(* IEC 61131-3 sources: test/Class/Sfc_Client_Splitter_4, 1 file *)

(* ---- Sfc_Client_Splitter_4.st ---- *)
(*!
<Class
	Name               = "Sfc_Client_Splitter_4"
	Revision           = "1.2"
	RealtimeTask       = "false"
	CyclicTask         = "false"
	BackgroundTask     = "false"
	Sigmatek           = "true"
	OSInterface        = "false"
	HighPriority       = "false"
	Automatic          = "false"
	UpdateMode         = "Prescan"
	IconPath           = ".\Class\Sfc_Client_Splitter_4\Client_Splitter_Base.ico"
	SharedCommandTable = "true"
	Objectsize         = "(284,120)"
	Comment            = "Splitter Class with 4 Clients">
	<Channels>
		<Client Name="Ch1" Required="false" Internal="false" Comment="Channel 1"/>
		<Client Name="Ch2" Required="false" Internal="false" Comment="Channel 2"/>
		<Client Name="Ch3" Required="false" Internal="false" Comment="Channel 3"/>
		<Client Name="Ch4" Required="false" Internal="false" Comment="Channel 4"/>
	</Channels>
	<RevDoku>
		<Owner Company="Sigmatek" Author="hötant"/>
		<Dokumentation Revision="1.2" Date="07.05.10" Author="hötant" Company="Sigmatek" Description="removed Server &quot;To_Split&quot; from derived Class&#13;&#10;(Server of BaseClass has the correct settings )"/>
	</RevDoku>
	<Network Name="Sfc_Client_Splitter_4">
		<!-- List of Components in this network -->
		<Components>
			<Object
				Name       = "_base"
				Class      = "Sfc_Client_Splitter_Base"
				Position   = "(1080,180)"
				Visualized = "false">
				<Channels>
					<Server Name="To_Splitt"/>
				</Channels>
			</Object>
		</Components>
		<Comments>
		</Comments>
		<!-- List of Connections in this network -->
		<Connections>
			<Connection Source="this.To_Splitt" Destination="_base.To_Splitt" Vertices="(1552,210),(1380,270),"/>
		</Connections>
		<!-- Headerfiles -->
		<Options>
		</Options>
	</Network>
</Class>
*)
#pragma using Sfc_Client_Splitter_Base

Sfc_Client_Splitter_4 : CLASS
: Sfc_Client_Splitter_Base
  //Servers:
  //Clients:
	Ch1 	: CltCh_DINT;
	Ch2 	: CltCh_DINT;
	Ch3 	: CltCh_DINT;
	Ch4 	: CltCh_DINT;
  //Variables:
  //Functions:
  //Tables:
	FUNCTION @STD
		VAR_OUTPUT
			ret_code	: CONFSTATES;
		END_VAR;
	FUNCTION GLOBAL TAB @CT_;
END_CLASS;
